FUNCTION_BLOCK Q_GraphicsContext (* Command Graphics Context ( Part 6 - F.56 ) *)
  (* Standard: ISO 11783-6; Description: This command is used to manipulate a graphics Context object (only on version 4 or later VTs). Return values iso_s16 - E_NO_ERR - OK - E_OVERFLOW - buffer overflow - E_NOACT - Command not possible in current state - E_NO_INSTANCE - No VT client available Note - Function uses string buffer ( Parameterlist has to be smaller than ISO_VTC_CMD_STR_MAX_LENGTH ) *)
  (* Version 1.0, 2022-07-08, franz *)
  (* Documentation:
  This command is used to manipulate a graphics Context object (only on version 4 or later VTs).
   Return values
   iso_s16
    - E_NO_ERR - OK
   - E_OVERFLOW - buffer overflow
   - E_NOACT - Command not possible in current state
   - E_NO_INSTANCE - No VT client available
    Note
    - Function uses string buffer ( Parameterlist has to be smaller than ISO_VTC_CMD_STR_MAX_LENGTH )
  *)
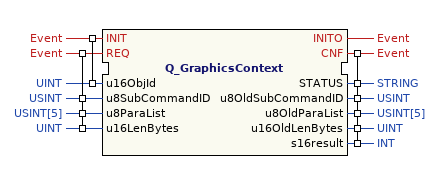
  EVENT_INPUT
    INIT WITH u16ObjId; (* Service Initialization *)
    REQ WITH u8SubCommandID, u8ParaList, u16LenBytes; (* Service Request *)
  END_EVENT
  EVENT_OUTPUT
    INITO; (* Initialization Confirm *)
    CNF WITH STATUS, s16result, u8OldSubCommandID, u8OldParaList, u16OldLenBytes; (* Confirmation of Requested Service *)
  END_EVENT
  VAR_INPUT
    u16ObjId : UINT; (* Object ID *)
    u8SubCommandID : USINT; (* Sub-Command ID *)
    u8ParaList : ARRAY [0..4] OF USINT; (* Parameters based on sub-command ID byte *)
    u16LenBytes : UINT; (* Length in bytes of parameter list *)
  END_VAR
  VAR_OUTPUT
    STATUS : STRING; (* Service Status *)
    u8OldSubCommandID : USINT; (* Old Sub-Command ID *)
    u8OldParaList : ARRAY [0..4] OF USINT; (* Old parameters based on sub-command ID byte *)
    u16OldLenBytes : UINT; (* Old length in bytes of parameter list *)
    s16result : INT; (* retval see description *)
  END_VAR
END_FUNCTION_BLOCK
